Omron CX-Programmer project NewProject (CX-Programmer 9.61)

# PLC Washing_Automatis: CP1L M

## Global symbols (name address type ; comment)
10.00 BOOL  ; MOTOR
0.00 BOOL  ; START
0.01 BOOL  ; STOP
0.02 BOOL  ; SENSOR
100.02 BOOL  ; BRUSH
10.01 BOOL  ; SPRAY
10.02 BOOL  ; BRUSH
1.00 BOOL  ; MOTOR
60.00 BOOL  ; IR
6.00 BOOL  ; IR

## Program NewProgram1 (cyclic task 0)

### Section Section1

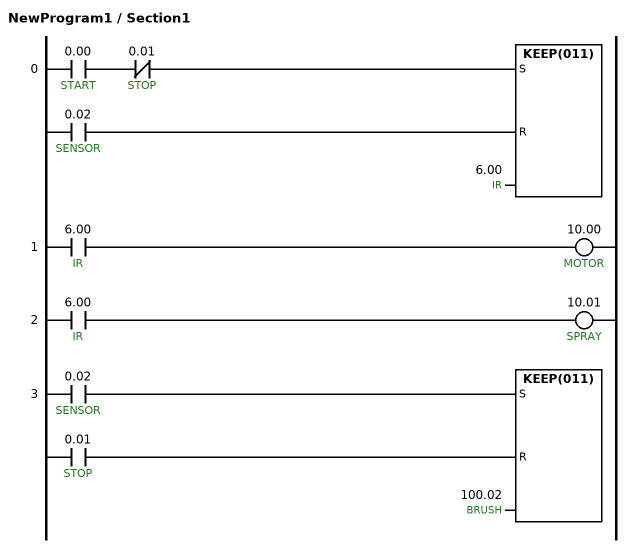
; rung 0
LD 0.00  ; START
ANDNOT 0.01  ; STOP
LD 0.02  ; SENSOR
KEEP(011) 6.00  ; IR
; rung 1
LD 6.00  ; IR
OUT 10.00  ; MOTOR
; rung 2
LD 6.00  ; IR
OUT 10.01  ; SPRAY
; rung 3
LD 0.02  ; SENSOR
LD 0.01  ; STOP
KEEP(011) 100.02  ; BRUSH

### Section END
; rung 0
END(001)